PROGRAM MAIN
VAR
	outer	: FB_Outer(Parameters.Parameters);
END_VAR

END_PROGRAM

(* stored: Version 1.1.0.1, ProductVersion 3.1.4024.15
   POU MAIN: Id {7d9634d2-d362-4e98-b674-0ec0eb263660}, SpecialFunc None *)
